{attribute addProperty BoxType "ER4374-0002-0018"}
{attribute addProperty Id "AI_Inputs_ChannelAT %I*ARRAY[0..2] OF AI_Inputs_Channel_087F71C76480AO_Outputs_ChannelAT %Q*ARRAY[0..1] OF AO_Outputs_Channel_F57FA4F93240WcStateAT %I*WcState_98A4DF7520.250InfoDataAT %I*InfoData_BC63D37F80100"}
{attribute addProperty CRC "3683339971"}
{attribute addProperty SizeInBites "178"}
{attribute addProperty SizeInBytes "22.25"}
TYPE ER4374_6989BFFB :
STRUCT
	{attribute addProperty Name "AI_Inputs_Channel"}
	AI_Inputs_Channel : ARRAY[0..2] OF AI_Inputs_Channel_087F71C7;
	{attribute addProperty Name "AO_Outputs_Channel"}
	AO_Outputs_Channel : ARRAY[0..1] OF AO_Outputs_Channel_F57FA4F9;
	{attribute addProperty Name "WcState"}
	WcState : WcState_98A4DF75;
	{attribute addProperty Name "InfoData"}
	InfoData : InfoData_BC63D37F;
END_STRUCT
END_TYPE

(* stored: Version 1.2.0.0, ProductVersion 3.1.4024.9
   DUT ER4374_6989BFFB: Id {fedacf4c-006a-48c6-a8be-d3698aaab8c8} *)
